// TIA Portal project "THITHU" (V14)

(* hardware
DEVICE "S7300/ET200M station_1"  S7-300 station
   slot 0: "Rail_0"  Rail  6ES7 390-1***0-0AA0
   slot 2: "PLC_1"  CPU 314C-2 PN/DP  6ES7 314-6EH04-0AB0  V3.3
      slot 2: "PROFINET interface_1"  PN-IO
         slot 1: "Port_1"  Port
         slot 2: "Port_2"  Port
      slot 5: "DI 24/DO 16_1"  DI24/DO16
      slot 6: "AI 5/AO 2_1"  AI5/AO2
      slot 7: "Count_1"  Counter
      slot 8: "Positioning_1"  Positioning
   slot 4: "DO 8x24VDC/2A_1"  DO8 x 24VDC / 2A  6ES7 322-1BF01-0AA0
*)

// ===== PLC "PLC_1"  CPU 314C-2 PN/DP =====

VAR_GLOBAL   // PLC tag table "Default tag table"
   "F5" AT %I0.0 : Bool;
   "S3" AT %I0.1 : Bool;
   "S4" AT %I0.2 : Bool;
   "S5" AT %I0.3 : Bool;
   "S6" AT %I0.4 : Bool;
   "S7" AT %I0.5 : Bool;
   "S8" AT %I0.6 : Bool;
   "S9" AT %I0.7 : Bool;
   "S10" AT %I1.0 : Bool;
   "S11" AT %I1.1 : Bool;
   "XX1" AT %I1.2 : Bool;
   "BP1" AT %I1.3 : Bool;
   "B1" AT %I1.4 : Bool;
   "B2" AT %I1.5 : Bool;
   "XX2" AT %I1.6 : Bool;
   "B11" AT %I1.7 : Bool;
   "B12" AT %I2.0 : Bool;
   "B21" AT %I2.1 : Bool;
   "B22" AT %I2.2 : Bool;
   "B31" AT %I2.3 : Bool;
   "B32" AT %I2.4 : Bool;
   "XX3" AT %I2.5 : Bool;
   "XX4" AT %I2.6 : Bool;
   "XX5" AT %I2.7 : Bool;
   "M11" AT %Q0.0 : Bool;
   "M12" AT %Q0.1 : Bool;
   "M21" AT %Q0.2 : Bool;
   "M22" AT %Q0.3 : Bool;
   "M31" AT %Q0.4 : Bool;
   "M32" AT %Q0.5 : Bool;
   "QQ1" AT %Q0.6 : Bool;
   "QQ2" AT %Q0.7 : Bool;
   "P32" AT %Q1.0 : Bool;
   "P33" AT %Q1.1 : Bool;
   "QQ3" AT %Q1.2 : Bool;
   "P2" AT %Q1.3 : Bool;
   "P3" AT %Q1.4 : Bool;
   "P4" AT %Q1.5 : Bool;
   "P5" AT %Q1.6 : Bool;
   "P6" AT %Q1.7 : Bool;
   "P7" AT %Q2.0 : Bool;
   "QQ4" AT %Q2.1 : Bool;
   "P10" AT %Q2.2 : Bool;
   "P11" AT %Q2.3 : Bool;
   "P12" AT %Q2.4 : Bool;
   "P13" AT %Q2.5 : Bool;
   "P14" AT %Q2.6 : Bool;
   "P15" AT %Q2.7 : Bool;
END_VAR

DATA_BLOCK "kich hoat toan he thong_DB"   // DB3
{ S7_Optimized_Access := 'FALSE' }
VERSION : 0.1
// stored: InstanceOfName kich hoat toan he thong
"kich hoat toan he thong"
BEGIN
END_DATA_BLOCK

DATA_BLOCK "THIET LAP AUTO/ TRUY VAN_DB"   // DB4
{ S7_Optimized_Access := 'FALSE' }
VERSION : 0.1
// stored: InstanceOfName THIET LAP AUTO/ TRUY VAN
"THIET LAP AUTO/ TRUY VAN"
BEGIN
END_DATA_BLOCK

DATA_BLOCK "NHAPNHAY_DB"   // DB5
{ S7_Optimized_Access := 'FALSE' }
VERSION : 0.1
// stored: InstanceOfName NHAPNHAY
"NHAPNHAY"
BEGIN
END_DATA_BLOCK

DATA_BLOCK "Manual_DB"   // DB6
{ S7_Optimized_Access := 'FALSE' }
VERSION : 0.1
// stored: InstanceOfName Manual
"Manual"
BEGIN
END_DATA_BLOCK

DATA_BLOCK "DEN BAO NHAN BIET_DB"   // DB7
{ S7_Optimized_Access := 'FALSE' }
VERSION : 0.1
// stored: InstanceOfName DEN BAO NHAN BIET
"DEN BAO NHAN BIET"
BEGIN
END_DATA_BLOCK

DATA_BLOCK "AUTO_DB"   // DB21
{ S7_Optimized_Access := 'FALSE' }
VERSION : 0.1
// stored: InstanceOfName AUTO
"AUTO"
BEGIN
END_DATA_BLOCK

DATA_BLOCK "OUTPUT_DB"   // DB22
{ S7_Optimized_Access := 'FALSE' }
VERSION : 0.1
// stored: InstanceOfName OUTPUT
"OUTPUT"
BEGIN
END_DATA_BLOCK

FUNCTION_BLOCK "kich hoat toan he thong"   // FB1, FBD
{ S7_Optimized_Access := 'FALSE' }
VERSION : 0.1
   VAR_INPUT
      F5 : Bool;
      BP1 : Bool;
      S3 : Bool;
      S4 : Bool;
      "KICH HOAT" : Bool;
   END_VAR
   VAR_OUTPUT
      "G-HIEN THI" : Bool;
      "CHI BAO VAN HANH" : Bool;
   END_VAR
   VAR
      X2 : Bool;
      X3 : Bool;
      X4 : Bool;
      X5 : Bool;
      X6 : Bool;
      p : Bool;
      X1 : Bool;
   END_VAR
   VAR_TEMP   // added for the SCL form of the ladder/FBD networks
      _w1 : Bool;
   END_VAR
BEGIN

REGION Network 1
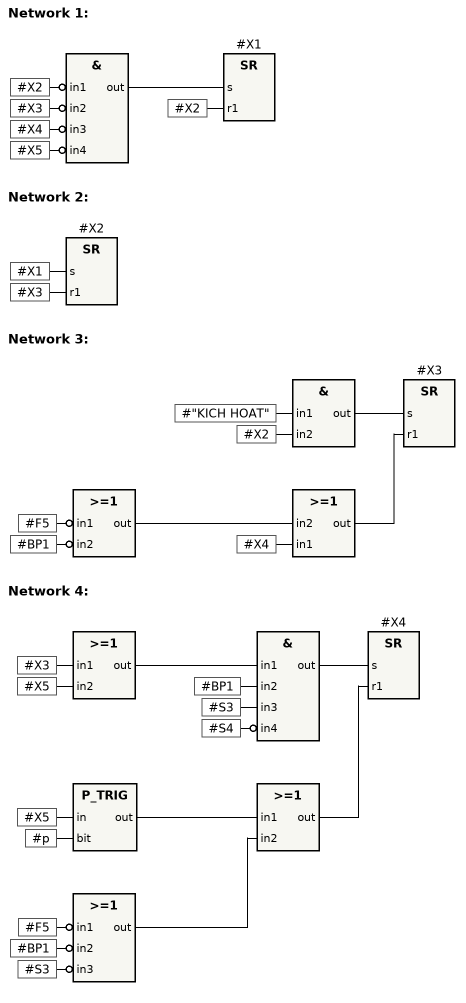
   IF NOT #X2 AND NOT #X3 AND NOT #X4 AND NOT #X5 THEN
       #X1 := TRUE;   // SR flip-flop
   END_IF;
   IF #X2 THEN #X1 := FALSE; END_IF;
END_REGION

REGION Network 2
   IF #X1 THEN
       #X2 := TRUE;   // SR flip-flop
   END_IF;
   IF #X3 THEN #X2 := FALSE; END_IF;
END_REGION

REGION Network 3
   IF #"KICH HOAT" AND #X2 THEN
       #X3 := TRUE;   // SR flip-flop
   END_IF;
   IF NOT #F5 OR NOT #BP1 OR #X4 THEN #X3 := FALSE; END_IF;
END_REGION

REGION Network 4
   #_w1 := #X5 AND NOT #p;   // rising edge
   #p := #X5;
   IF (#X3 OR #X5) AND #BP1 AND #S3 AND NOT #S4 THEN
       #X4 := TRUE;   // SR flip-flop
   END_IF;
   IF #_w1 OR NOT #F5 OR NOT #BP1 OR NOT #S3 THEN #X4 := FALSE; END_IF;
END_REGION

REGION Network 5
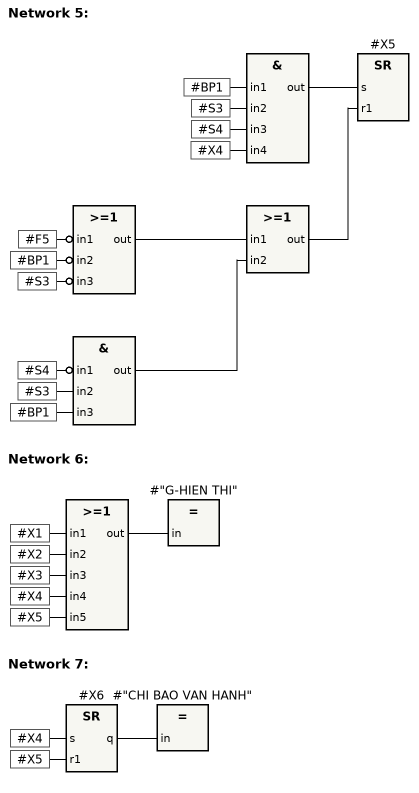
   IF #BP1 AND #S3 AND #S4 AND #X4 THEN
       #X5 := TRUE;   // SR flip-flop
   END_IF;
   IF NOT #F5 OR NOT #BP1 OR NOT #S3 OR (NOT #S4 AND #S3 AND #BP1) THEN #X5 := FALSE; END_IF;
END_REGION

REGION Network 6
   #"G-HIEN THI" := #X1 OR #X2 OR #X3 OR #X4 OR #X5;
END_REGION

REGION Network 7
   IF #X4 THEN
       #X6 := TRUE;   // SR flip-flop
   END_IF;
   IF #X5 THEN #X6 := FALSE; END_IF;
   #"CHI BAO VAN HANH" := #X6;
END_REGION
END_FUNCTION_BLOCK

FUNCTION_BLOCK "NHAPNHAY"   // FB2, FBD
{ S7_Optimized_Access := 'FALSE' }
VERSION : 0.1
   VAR_OUTPUT
      BUOC : Bool;
   END_VAR
   VAR
      X1 : Bool;
      X2 : Bool;
      X3 : Bool;
      X4 : Bool;
   END_VAR
BEGIN

REGION Network 1
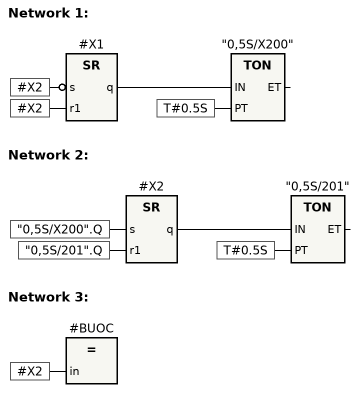
   IF NOT #X2 THEN
       #X1 := TRUE;   // SR flip-flop
   END_IF;
   IF #X2 THEN #X1 := FALSE; END_IF;
   "0,5S/X200".TON(IN := #X1, PT := T#0.5S);
END_REGION

REGION Network 2
   IF "0,5S/X200".Q THEN
       #X2 := TRUE;   // SR flip-flop
   END_IF;
   IF "0,5S/201".Q THEN #X2 := FALSE; END_IF;
   "0,5S/201".TON(IN := #X2, PT := T#0.5S);
END_REGION

REGION Network 3
   #BUOC := #X2;
END_REGION
END_FUNCTION_BLOCK

FUNCTION_BLOCK "THIET LAP AUTO/ TRUY VAN"   // FB3, FBD
{ S7_Optimized_Access := 'FALSE' }
VERSION : 0.1
   VAR_INPUT
      F5 : Bool;
      S3 : Bool;
      S4 : Bool;
      S5 : Bool;
      S6 : Bool;
      S7 : Bool;
      S8 : Bool;
      S9 : Bool;
      S10 : Bool;
      "G-KICH HOAT" : Bool;
      S11 : Bool;
   END_VAR
   VAR_OUTPUT
      P32 : Bool;
      P6 : Bool;
      "KICH HOAT" : Bool;
      P33 : Bool;
   END_VAR
   VAR
      X1 : Bool;
      X2 : Bool;
      X3 : Bool;
      X4 : Bool;
      X5 : Bool;
      X6 : Bool;
   END_VAR
BEGIN

REGION Network 1
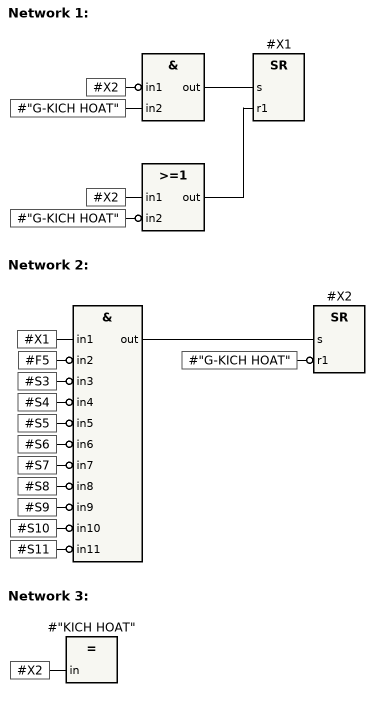
   IF NOT #X2 AND #"G-KICH HOAT" THEN
       #X1 := TRUE;   // SR flip-flop
   END_IF;
   IF #X2 OR NOT #"G-KICH HOAT" THEN #X1 := FALSE; END_IF;
END_REGION

REGION Network 2
   IF #X1 AND NOT #F5 AND NOT #S3 AND NOT #S4 AND NOT #S5 AND NOT #S6 AND NOT #S7 AND NOT #S8 AND NOT #S9 AND NOT #S10 AND NOT #S11 THEN
       #X2 := TRUE;   // SR flip-flop
   END_IF;
   IF NOT #"G-KICH HOAT" THEN #X2 := FALSE; END_IF;
END_REGION

REGION Network 3
   #"KICH HOAT" := #X2;
END_REGION
END_FUNCTION_BLOCK

FUNCTION_BLOCK "Manual"   // FB4, FBD
{ S7_Optimized_Access := 'FALSE' }
VERSION : 0.1
   VAR_INPUT
      S6 : Bool;
      S7 : Bool;
      S8 : Bool;
      S9 : Bool;
      S10 : Bool;
      S11 : Bool;
      B11 : Bool;
      B12 : Bool;
      B21 : Bool;
      B22 : Bool;
      B31 : Bool;
      "G-Manual" : Bool;
      B32 : Bool;
   END_VAR
   VAR_OUTPUT
      M11 : Bool;
      M12 : Bool;
      M21 : Bool;
      M22 : Bool;
      M31 : Bool;
      M32 : Bool;
   END_VAR
   VAR
      X1 : Bool;
      X2 : Bool;
      X3 : Bool;
      X4 : Bool;
      X5 : Bool;
   END_VAR
BEGIN

REGION Network 1
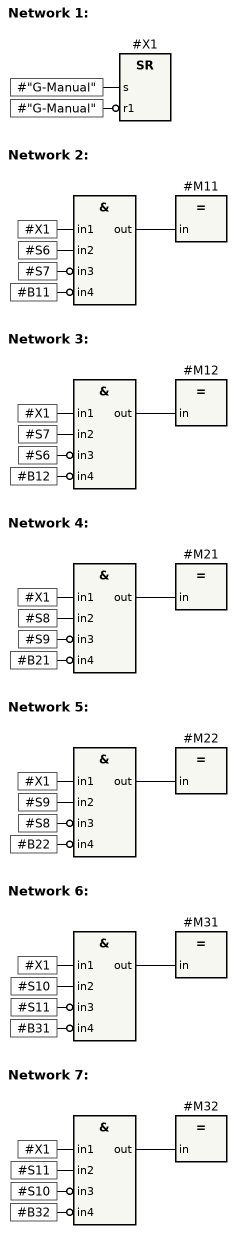
   IF #"G-Manual" THEN
       #X1 := TRUE;   // SR flip-flop
   END_IF;
   IF NOT #"G-Manual" THEN #X1 := FALSE; END_IF;
END_REGION

REGION Network 2
   #M11 := #X1 AND #S6 AND NOT #S7 AND NOT #B11;
END_REGION

REGION Network 3
   #M12 := #X1 AND #S7 AND NOT #S6 AND NOT #B12;
END_REGION

REGION Network 4
   #M21 := #X1 AND #S8 AND NOT #S9 AND NOT #B21;
END_REGION

REGION Network 5
   #M22 := #X1 AND #S9 AND NOT #S8 AND NOT #B22;
END_REGION

REGION Network 6
   #M31 := #X1 AND #S10 AND NOT #S11 AND NOT #B31;
END_REGION

REGION Network 7
   #M32 := #X1 AND #S11 AND NOT #S10 AND NOT #B32;
END_REGION
END_FUNCTION_BLOCK

FUNCTION_BLOCK "DEN BAO NHAN BIET"   // FB5, FBD
{ S7_Optimized_Access := 'FALSE' }
VERSION : 0.1
   VAR_INPUT
      S3 : Bool;
      B12 : Bool;
      B11 : Bool;
      B21 : Bool;
      B22 : Bool;
      B31 : Bool;
      B32 : Bool;
      B1 : Bool;
      BP1 : Bool;
      B2 : Bool;
      BUOC : Bool;
      "G-hien thi" : Bool;
      "CHI BAO VAN HANH" : Bool;
   END_VAR
   VAR_OUTPUT
      P2 : Bool;
      P3 : Bool;
      P4 : Bool;
      P7 : Bool;
      P10 : Bool;
      P11 : Bool;
      P12 : Bool;
      P13 : Bool;
      P14 : Bool;
      P15 : Bool;
   END_VAR
   VAR
      X1 : Bool;
      X2 : Bool;
      X3 : Bool;
      X4 : Bool;
      X5 : Bool;
      X6 : Bool;
   END_VAR
BEGIN

REGION Network 1
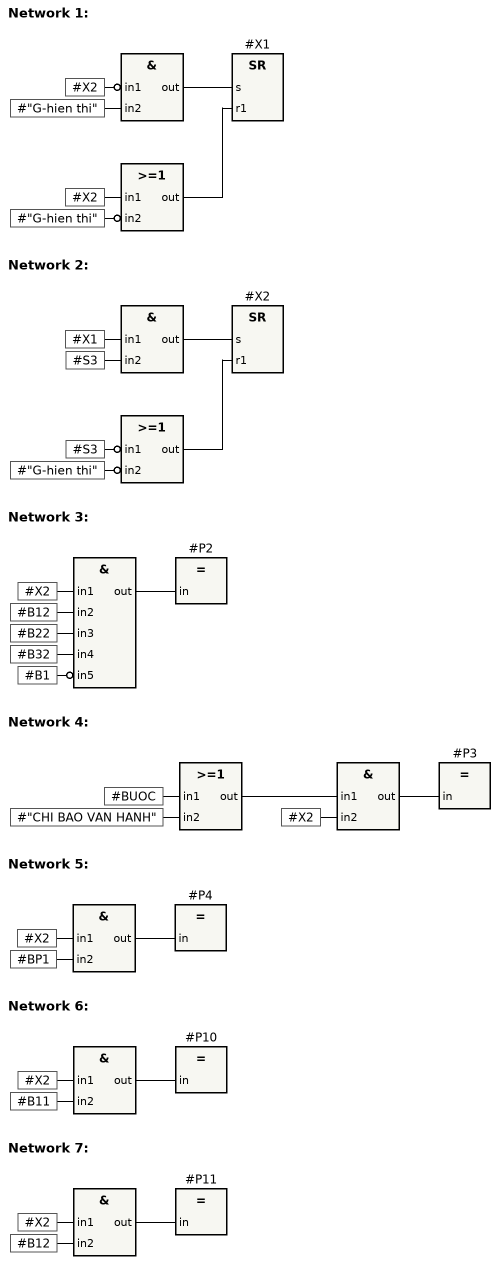
   IF NOT #X2 AND #"G-hien thi" THEN
       #X1 := TRUE;   // SR flip-flop
   END_IF;
   IF #X2 OR NOT #"G-hien thi" THEN #X1 := FALSE; END_IF;
END_REGION

REGION Network 2
   IF #X1 AND #S3 THEN
       #X2 := TRUE;   // SR flip-flop
   END_IF;
   IF NOT #S3 OR NOT #"G-hien thi" THEN #X2 := FALSE; END_IF;
END_REGION

REGION Network 3
   #P2 := #X2 AND #B12 AND #B22 AND #B32 AND NOT #B1;
END_REGION

REGION Network 4
   #P3 := (#BUOC OR #"CHI BAO VAN HANH") AND #X2;
END_REGION

REGION Network 5
   #P4 := #X2 AND #BP1;
END_REGION

REGION Network 6
   #P10 := #X2 AND #B11;
END_REGION

REGION Network 7
   #P11 := #X2 AND #B12;
END_REGION

REGION Network 8
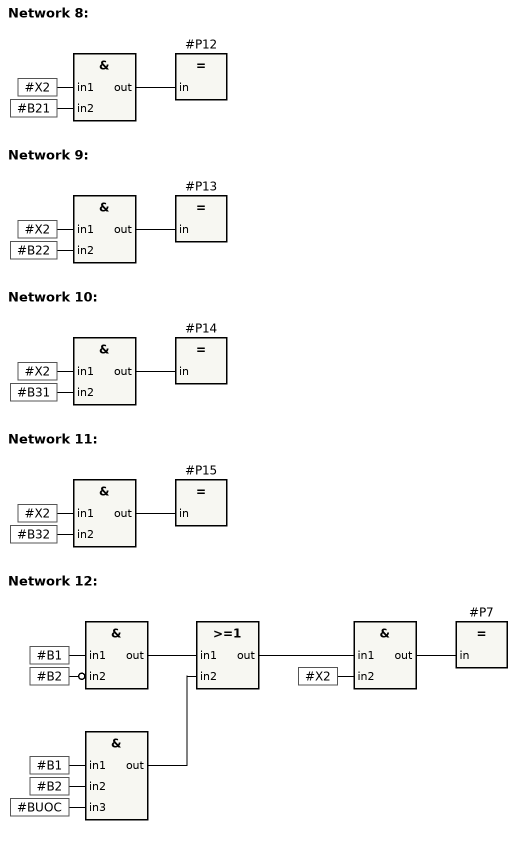
   #P12 := #X2 AND #B21;
END_REGION

REGION Network 9
   #P13 := #X2 AND #B22;
END_REGION

REGION Network 10
   #P14 := #X2 AND #B31;
END_REGION

REGION Network 11
   #P15 := #X2 AND #B32;
END_REGION

REGION Network 12
   #P7 := ((#B1 AND NOT #B2) OR (#B1 AND #B2 AND #BUOC)) AND #X2;
END_REGION
END_FUNCTION_BLOCK

FUNCTION_BLOCK "AUTO"   // FB6, FBD
{ S7_Optimized_Access := 'FALSE' }
VERSION : 0.1
   VAR_INPUT
      S5 : Bool;
      B11 : Bool;
      B12 : Bool;
      B21 : Bool;
      B31 : Bool;
      B1 : Bool;
      "G-AUTO" : Bool;
      P2 : Bool;
      X50 : Bool;
      "CHI BAO VAN HANH" : Bool;
      B2 : Bool;
   END_VAR
   VAR_OUTPUT
      P32 : Bool;
      P33 : Bool;
      M11 : Bool;
      M12 : Bool;
      M21 : Bool;
      M22 : Bool;
      M31 : Bool;
      P5 : Bool;
      P6 : Bool;
      M32 : Bool;
   END_VAR
   VAR
      X60 : Bool;
      X61 : Bool;
      X62 : Bool;
      X63 : Bool;
      X64a : Bool;
      X64 : Bool;
      X65 : Bool;
      X66 : Bool;
      X67 : Bool;
      X68 : Bool;
      X69 : Bool;
      "PHOI CO" : Bool;
      P : Bool;
      X1 : Bool;
      X2 : Bool;
      X3 : Bool;
      X4 : Bool;
      X5 : Bool;
      X6 : Bool;
      X7 : Bool;
   END_VAR
   VAR_TEMP   // added for the SCL form of the ladder/FBD networks
      _w1 : Bool;
   END_VAR
BEGIN

REGION Network 1
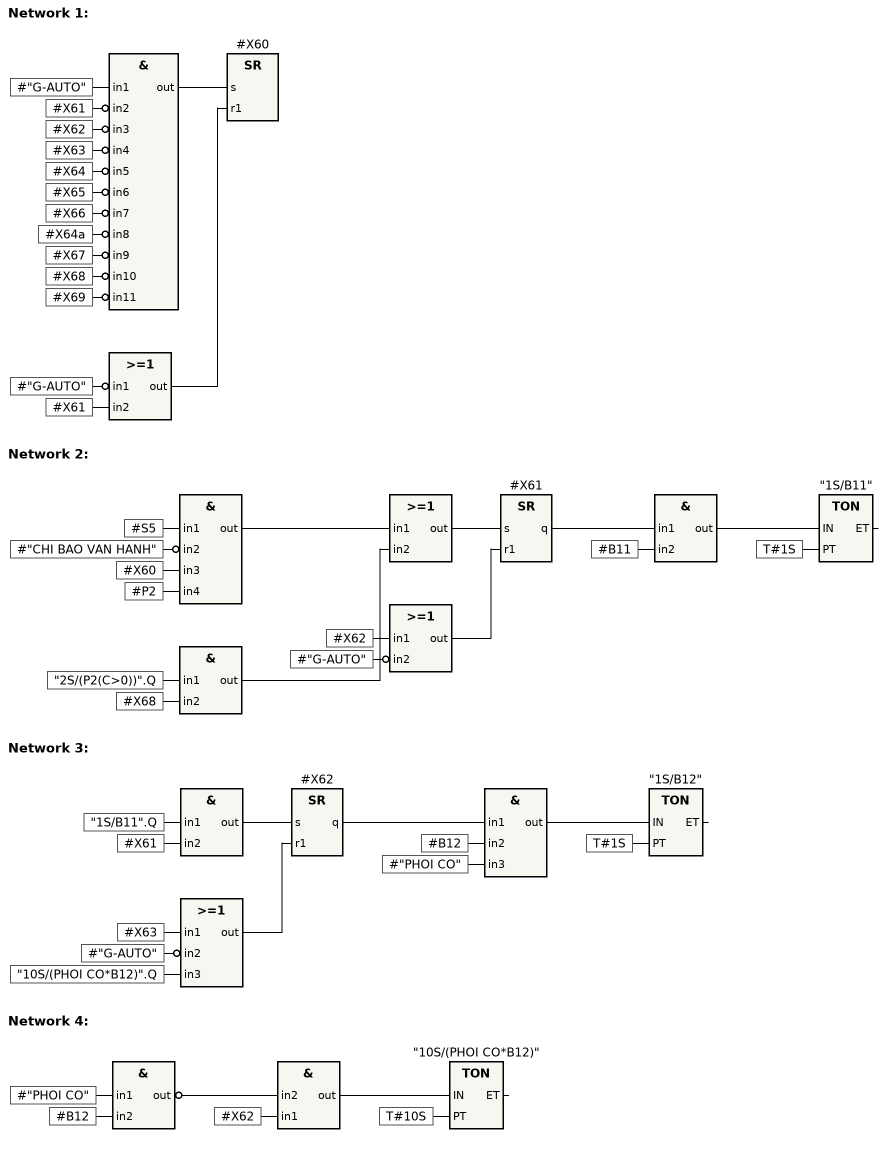
   IF #"G-AUTO" AND NOT #X61 AND NOT #X62 AND NOT #X63 AND NOT #X64 AND NOT #X65 AND NOT #X66 AND NOT #X64a AND NOT #X67 AND NOT #X68 AND NOT #X69 THEN
       #X60 := TRUE;   // SR flip-flop
   END_IF;
   IF NOT #"G-AUTO" OR #X61 THEN #X60 := FALSE; END_IF;
END_REGION

REGION Network 2
   IF (#S5 AND NOT #"CHI BAO VAN HANH" AND #X60 AND #P2) OR ("2S/(P2(C>0))".Q AND #X68) THEN
       #X61 := TRUE;   // SR flip-flop
   END_IF;
   IF #X62 OR NOT #"G-AUTO" THEN #X61 := FALSE; END_IF;
   "1S/B11".TON(IN := #X61 AND #B11, PT := T#1S);
END_REGION

REGION Network 3
   IF "1S/B11".Q AND #X61 THEN
       #X62 := TRUE;   // SR flip-flop
   END_IF;
   IF #X63 OR NOT #"G-AUTO" OR "10S/(PHOI CO*B12)".Q THEN #X62 := FALSE; END_IF;
   "1S/B12".TON(IN := #X62 AND #B12 AND #"PHOI CO", PT := T#1S);
END_REGION

REGION Network 4
   "10S/(PHOI CO*B12)".TON(IN := NOT (#"PHOI CO" AND #B12) AND #X62, PT := T#10S);
END_REGION

REGION Network 5
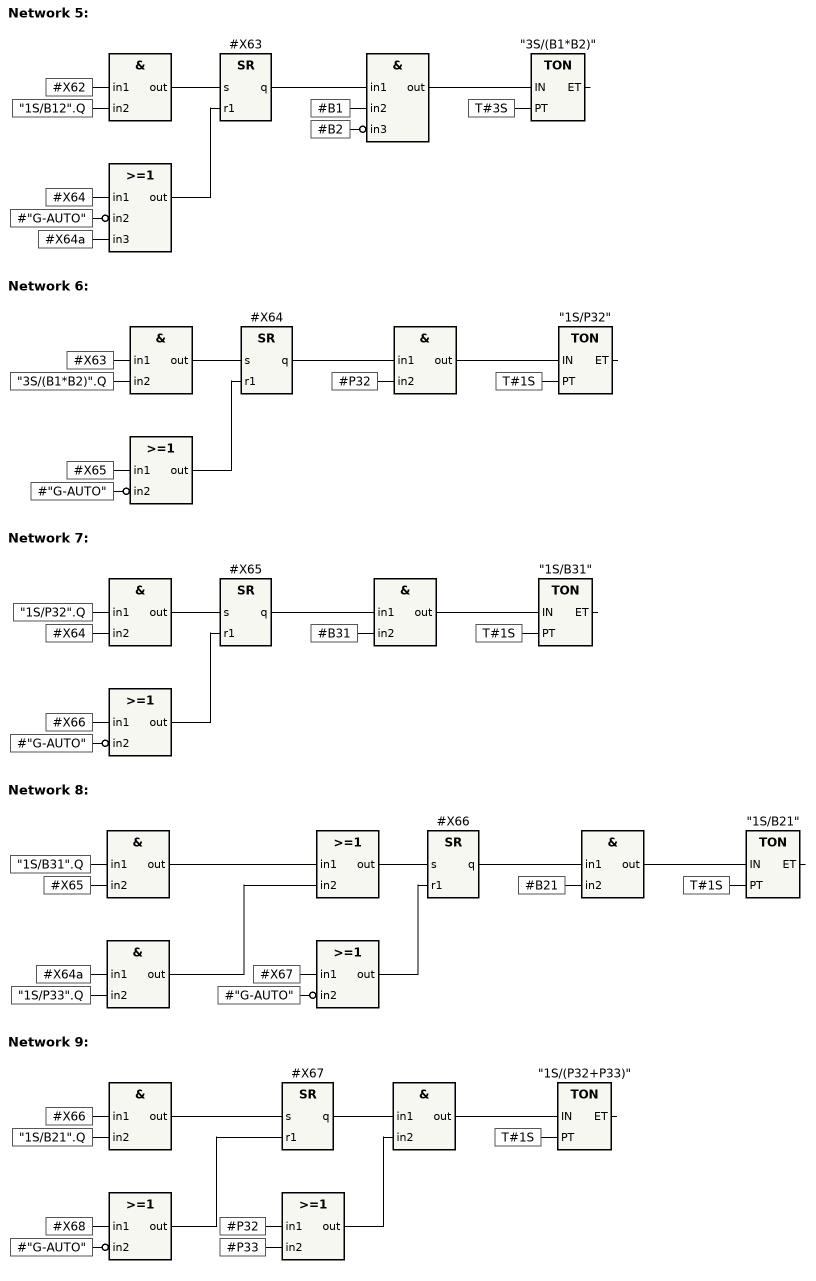
   IF #X62 AND "1S/B12".Q THEN
       #X63 := TRUE;   // SR flip-flop
   END_IF;
   IF #X64 OR NOT #"G-AUTO" OR #X64a THEN #X63 := FALSE; END_IF;
   "3S/(B1*B2)".TON(IN := #X63 AND #B1 AND NOT #B2, PT := T#3S);
END_REGION

REGION Network 6
   IF #X63 AND "3S/(B1*B2)".Q THEN
       #X64 := TRUE;   // SR flip-flop
   END_IF;
   IF #X65 OR NOT #"G-AUTO" THEN #X64 := FALSE; END_IF;
   "1S/P32".TON(IN := #X64 AND #P32, PT := T#1S);
END_REGION

REGION Network 7
   IF "1S/P32".Q AND #X64 THEN
       #X65 := TRUE;   // SR flip-flop
   END_IF;
   IF #X66 OR NOT #"G-AUTO" THEN #X65 := FALSE; END_IF;
   "1S/B31".TON(IN := #X65 AND #B31, PT := T#1S);
END_REGION

REGION Network 8
   IF ("1S/B31".Q AND #X65) OR (#X64a AND "1S/P33".Q) THEN
       #X66 := TRUE;   // SR flip-flop
   END_IF;
   IF #X67 OR NOT #"G-AUTO" THEN #X66 := FALSE; END_IF;
   "1S/B21".TON(IN := #X66 AND #B21, PT := T#1S);
END_REGION

REGION Network 9
   IF #X66 AND "1S/B21".Q THEN
       #X67 := TRUE;   // SR flip-flop
   END_IF;
   IF #X68 OR NOT #"G-AUTO" THEN #X67 := FALSE; END_IF;
   "1S/(P32+P33)".TON(IN := #X67 AND (#P32 OR #P33), PT := T#1S);
END_REGION

REGION Network 10
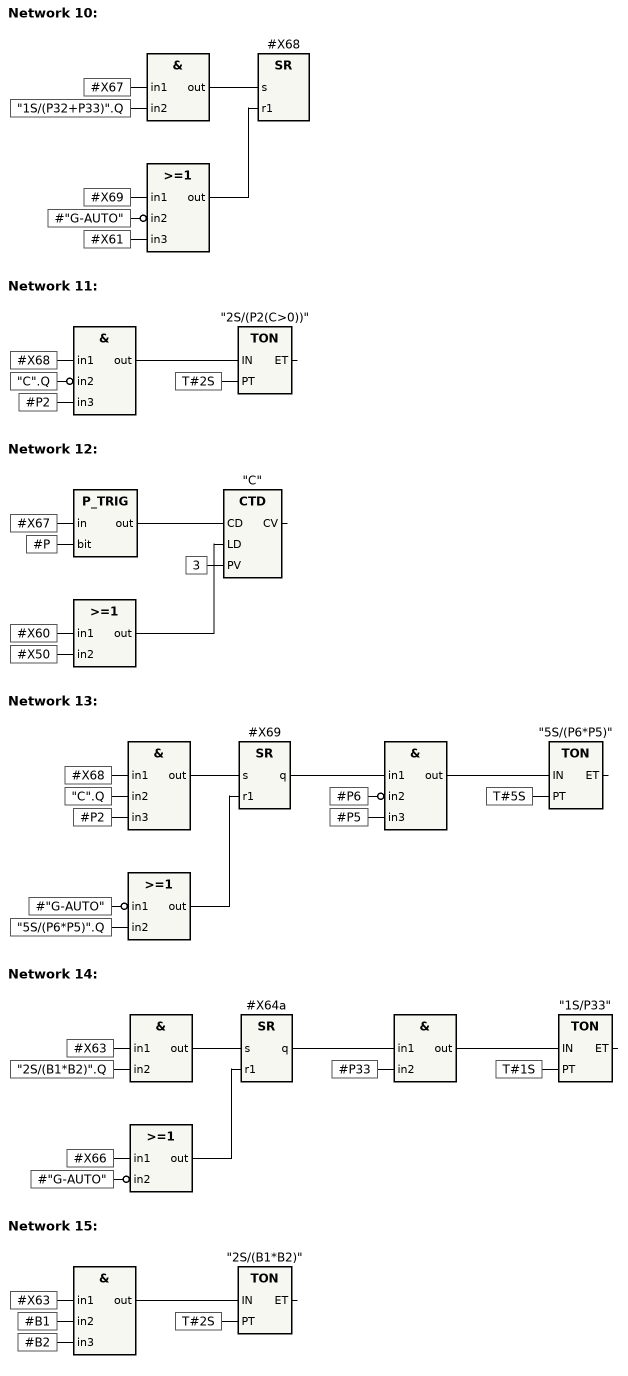
   IF #X67 AND "1S/(P32+P33)".Q THEN
       #X68 := TRUE;   // SR flip-flop
   END_IF;
   IF #X69 OR NOT #"G-AUTO" OR #X61 THEN #X68 := FALSE; END_IF;
END_REGION

REGION Network 11
   "2S/(P2(C>0))".TON(IN := #X68 AND NOT "C".Q AND #P2, PT := T#2S);
END_REGION

REGION Network 12
   #_w1 := #X67 AND NOT #P;   // rising edge
   #P := #X67;
   "C".CTD(CD := #_w1, LD := #X60 OR #X50, PV := 3);
END_REGION

REGION Network 13
   IF #X68 AND "C".Q AND #P2 THEN
       #X69 := TRUE;   // SR flip-flop
   END_IF;
   IF NOT #"G-AUTO" OR "5S/(P6*P5)".Q THEN #X69 := FALSE; END_IF;
   "5S/(P6*P5)".TON(IN := #X69 AND NOT #P6 AND #P5, PT := T#5S);
END_REGION

REGION Network 14
   IF #X63 AND "2S/(B1*B2)".Q THEN
       #X64a := TRUE;   // SR flip-flop
   END_IF;
   IF #X66 OR NOT #"G-AUTO" THEN #X64a := FALSE; END_IF;
   "1S/P33".TON(IN := #X64a AND #P33, PT := T#1S);
END_REGION

REGION Network 15
   "2S/(B1*B2)".TON(IN := #X63 AND #B1 AND #B2, PT := T#2S);
END_REGION

REGION Network 16
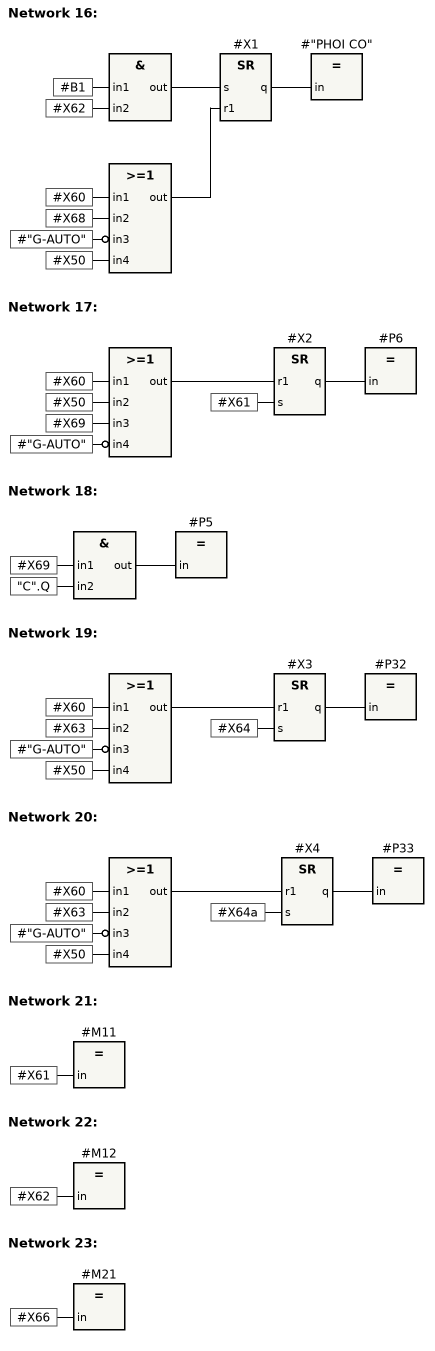
   IF #B1 AND #X62 THEN
       #X1 := TRUE;   // SR flip-flop
   END_IF;
   IF #X60 OR #X68 OR NOT #"G-AUTO" OR #X50 THEN #X1 := FALSE; END_IF;
   #"PHOI CO" := #X1;
END_REGION

REGION Network 17
   IF #X61 THEN
       #X2 := TRUE;   // SR flip-flop
   END_IF;
   IF #X60 OR #X50 OR #X69 OR NOT #"G-AUTO" THEN #X2 := FALSE; END_IF;
   #P6 := #X2;
END_REGION

REGION Network 18
   #P5 := #X69 AND "C".Q;
END_REGION

REGION Network 19
   IF #X64 THEN
       #X3 := TRUE;   // SR flip-flop
   END_IF;
   IF #X60 OR #X63 OR NOT #"G-AUTO" OR #X50 THEN #X3 := FALSE; END_IF;
   #P32 := #X3;
END_REGION

REGION Network 20
   IF #X64a THEN
       #X4 := TRUE;   // SR flip-flop
   END_IF;
   IF #X60 OR #X63 OR NOT #"G-AUTO" OR #X50 THEN #X4 := FALSE; END_IF;
   #P33 := #X4;
END_REGION

REGION Network 21
   #M11 := #X61;
END_REGION

REGION Network 22
   #M12 := #X62;
END_REGION

REGION Network 23
   #M21 := #X66;
END_REGION

REGION Network 24
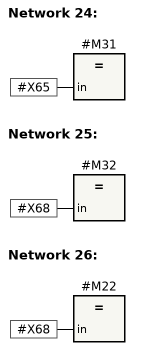
   #M31 := #X65;
END_REGION

REGION Network 25
   #M32 := #X68;
END_REGION

REGION Network 26
   #M22 := #X68;
END_REGION
END_FUNCTION_BLOCK

FUNCTION_BLOCK "OUTPUT"   // FB7, FBD
{ S7_Optimized_Access := 'FALSE' }
VERSION : 0.1
   VAR_INPUT
      M11_A : Bool;
      M11_M : Bool;
      M12_A : Bool;
      M12_M : Bool;
      M21_A : Bool;
      M21_M : Bool;
      M22_A : Bool;
      M22_M : Bool;
      M31_M : Bool;
      M32_A : Bool;
      M31_A : Bool;
      M32_M : Bool;
   END_VAR
   VAR_OUTPUT
      M11 : Bool;
      M12 : Bool;
      M21 : Bool;
      M22 : Bool;
      M31 : Bool;
      M32 : Bool;
   END_VAR
   VAR
      X1 : Bool;
      X2 : Bool;
      X3 : Bool;
      X4 : Bool;
      X5 : Bool;
      X6 : Bool;
   END_VAR
BEGIN

REGION Network 1
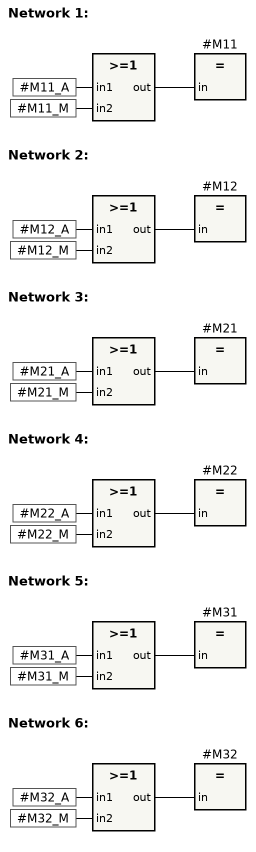
   #M11 := #M11_A OR #M11_M;
END_REGION

REGION Network 2
   #M12 := #M12_A OR #M12_M;
END_REGION

REGION Network 3
   #M21 := #M21_A OR #M21_M;
END_REGION

REGION Network 4
   #M22 := #M22_A OR #M22_M;
END_REGION

REGION Network 5
   #M31 := #M31_A OR #M31_M;
END_REGION

REGION Network 6
   #M32 := #M32_A OR #M32_M;
END_REGION
END_FUNCTION_BLOCK

ORGANIZATION_BLOCK "Main"   // OB1, FBD
TITLE = "Main Program Sweep (Cycle)"
{ S7_Optimized_Access := 'FALSE' }
VERSION : 0.1
   VAR_TEMP
      OB1_EV_CLASS : Byte;   // Bits 0-3 = 1 (Coming event), Bits 4-7 = 1 (Event class 1)
      OB1_SCAN_1 : Byte;   // 1 (Cold restart scan 1 of OB 1), 3 (Scan 2-n of OB 1)
      OB1_PRIORITY : Byte;   // Priority of OB Execution
      OB1_OB_NUMBR : Byte;   // 1 (Organization block 1, OB1)
      OB1_RESERVED_1 : Byte;   // Reserved for system
      OB1_RESERVED_2 : Byte;   // Reserved for system
      OB1_PREV_CYCLE : Int;   // Cycle time of previous OB1 scan (milliseconds)
      OB1_MIN_CYCLE : Int;   // Minimum cycle time of OB1 (milliseconds)
      OB1_MAX_CYCLE : Int;   // Maximum cycle time of OB1 (milliseconds)
      OB1_DATE_TIME : Date_And_Time;   // Date and time OB1 started
   END_VAR
BEGIN

REGION Network 1
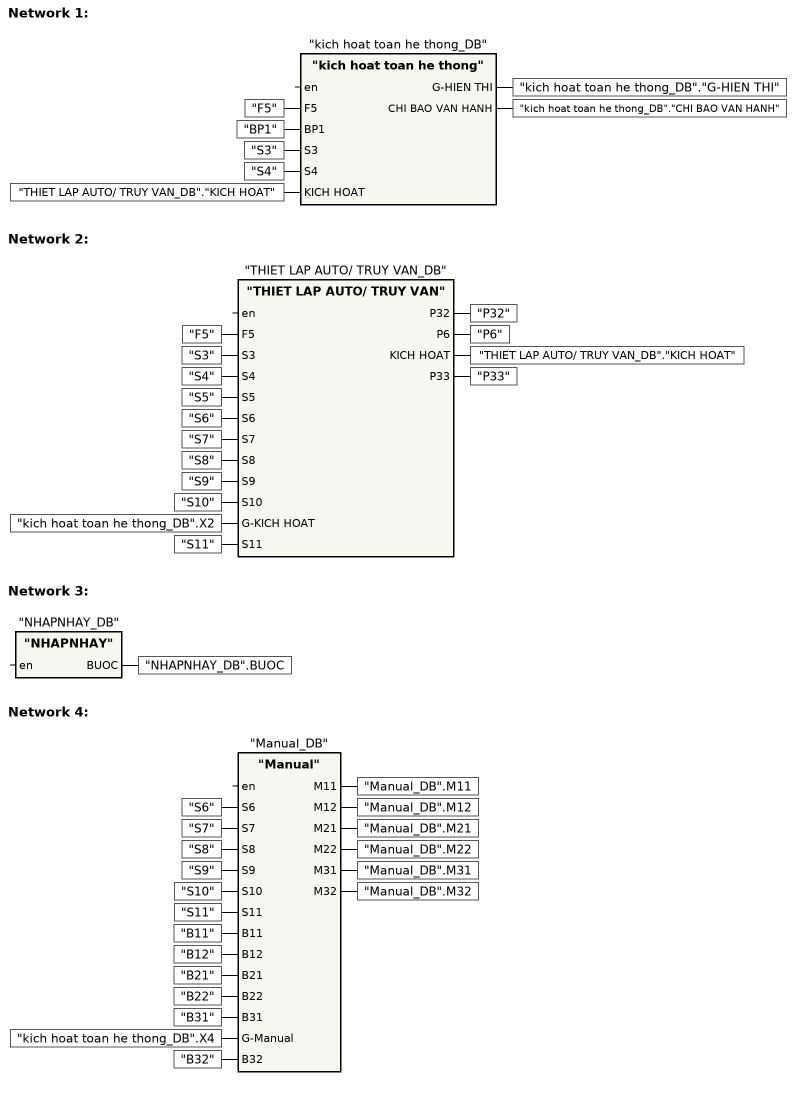
   "kich hoat toan he thong_DB"(F5 := "F5",   // "kich hoat toan he thong"
                           BP1 := "BP1",
                           S3 := "S3",
                           S4 := "S4",
                           "KICH HOAT" := "THIET LAP AUTO/ TRUY VAN_DB"."KICH HOAT",
                           "G-HIEN THI" => "kich hoat toan he thong_DB"."G-HIEN THI",
                           "CHI BAO VAN HANH" => "kich hoat toan he thong_DB"."CHI BAO VAN HANH");
END_REGION

REGION Network 2
   "THIET LAP AUTO/ TRUY VAN_DB"(F5 := "F5",   // "THIET LAP AUTO/ TRUY VAN"
                           S3 := "S3",
                           S4 := "S4",
                           S5 := "S5",
                           S6 := "S6",
                           S7 := "S7",
                           S8 := "S8",
                           S9 := "S9",
                           S10 := "S10",
                           "G-KICH HOAT" := "kich hoat toan he thong_DB".X2,
                           S11 := "S11",
                           P32 => "P32",
                           P6 => "P6",
                           "KICH HOAT" => "THIET LAP AUTO/ TRUY VAN_DB"."KICH HOAT",
                           P33 => "P33");
END_REGION

REGION Network 3
   "NHAPNHAY_DB"(BUOC => "NHAPNHAY_DB".BUOC);   // "NHAPNHAY"
END_REGION

REGION Network 4
   "Manual_DB"(S6 := "S6",   // "Manual"
               S7 := "S7",
               S8 := "S8",
               S9 := "S9",
               S10 := "S10",
               S11 := "S11",
               B11 := "B11",
               B12 := "B12",
               B21 := "B21",
               B22 := "B22",
               B31 := "B31",
               "G-Manual" := "kich hoat toan he thong_DB".X4,
               B32 := "B32",
               M11 => "Manual_DB".M11,
               M12 => "Manual_DB".M12,
               M21 => "Manual_DB".M21,
               M22 => "Manual_DB".M22,
               M31 => "Manual_DB".M31,
               M32 => "Manual_DB".M32);
END_REGION

REGION Network 5
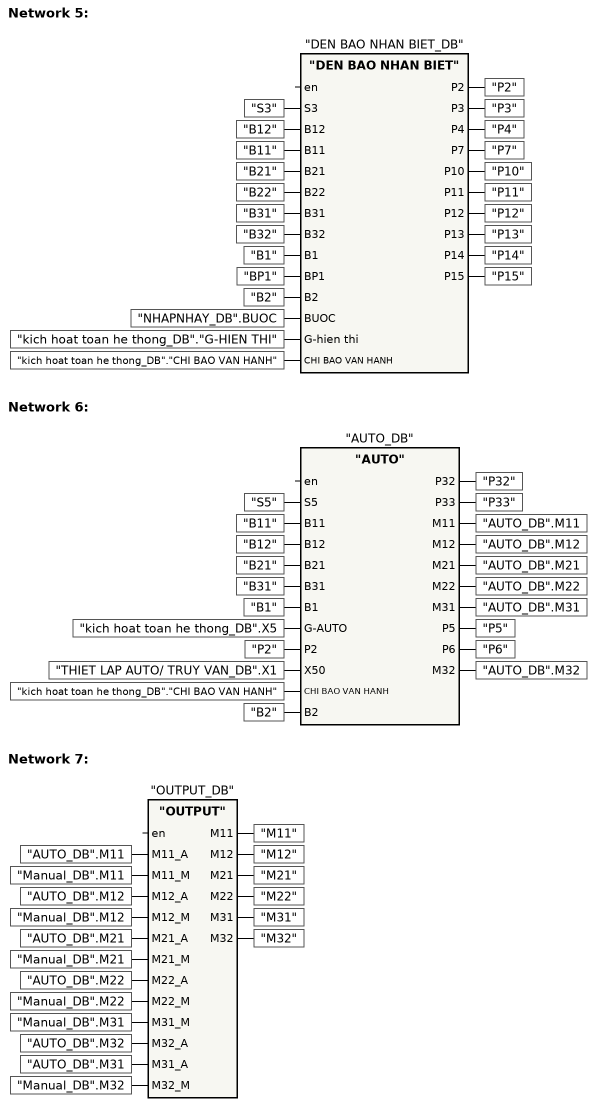
   "DEN BAO NHAN BIET_DB"(S3 := "S3",   // "DEN BAO NHAN BIET"
                          B12 := "B12",
                          B11 := "B11",
                          B21 := "B21",
                          B22 := "B22",
                          B31 := "B31",
                          B32 := "B32",
                          B1 := "B1",
                          BP1 := "BP1",
                          B2 := "B2",
                          BUOC := "NHAPNHAY_DB".BUOC,
                          "G-hien thi" := "kich hoat toan he thong_DB"."G-HIEN THI",
                          "CHI BAO VAN HANH" := "kich hoat toan he thong_DB"."CHI BAO VAN HANH",
                          P2 => "P2",
                          P3 => "P3",
                          P4 => "P4",
                          P7 => "P7",
                          P10 => "P10",
                          P11 => "P11",
                          P12 => "P12",
                          P13 => "P13",
                          P14 => "P14",
                          P15 => "P15");
END_REGION

REGION Network 6
   "AUTO_DB"(S5 := "S5",   // "AUTO"
             B11 := "B11",
             B12 := "B12",
             B21 := "B21",
             B31 := "B31",
             B1 := "B1",
             "G-AUTO" := "kich hoat toan he thong_DB".X5,
             P2 := "P2",
             X50 := "THIET LAP AUTO/ TRUY VAN_DB".X1,
             "CHI BAO VAN HANH" := "kich hoat toan he thong_DB"."CHI BAO VAN HANH",
             B2 := "B2",
             P32 => "P32",
             P33 => "P33",
             M11 => "AUTO_DB".M11,
             M12 => "AUTO_DB".M12,
             M21 => "AUTO_DB".M21,
             M22 => "AUTO_DB".M22,
             M31 => "AUTO_DB".M31,
             P5 => "P5",
             P6 => "P6",
             M32 => "AUTO_DB".M32);
END_REGION

REGION Network 7
   "OUTPUT_DB"(M11_A := "AUTO_DB".M11,   // "OUTPUT"
               M11_M := "Manual_DB".M11,
               M12_A := "AUTO_DB".M12,
               M12_M := "Manual_DB".M12,
               M21_A := "AUTO_DB".M21,
               M21_M := "Manual_DB".M21,
               M22_A := "AUTO_DB".M22,
               M22_M := "Manual_DB".M22,
               M31_M := "Manual_DB".M31,
               M32_A := "AUTO_DB".M32,
               M31_A := "AUTO_DB".M31,
               M32_M := "Manual_DB".M32,
               M11 => "M11",
               M12 => "M12",
               M21 => "M21",
               M22 => "M22",
               M31 => "M31",
               M32 => "M32");
END_REGION
END_ORGANIZATION_BLOCK